SUBAPPLICATION Uebung_10c4 (* SoftKey_F1/_F2 auf DigitalOutput_Q1/_Q2 mit GreenWhiteBackground mit Typed Subapp *)
  (* Standard: 61499-2; Description: Copyright (c) 2023 Meisterschulen am Ostbahnhof This program and the accompanying materials are made available under the terms of the Eclipse Public License 2.0 which is available at https://www.eclipse.org/legal/epl-2.0/ SPDX-License-Identifier: EPL-2.0 *)
  (* Version 1.0, 2023-10-23, Franz Höpfinger, Meisterschulen am Ostbahnhof *)
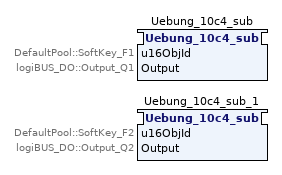
  SUBAPPS
    Uebung_10c4_sub : Uebung_10c4_sub(u16ObjId := DefaultPool::SoftKey_F1, Output := logiBUS_DO::Output_Q1);
    Uebung_10c4_sub_1 : Uebung_10c4_sub(u16ObjId := DefaultPool::SoftKey_F2, Output := logiBUS_DO::Output_Q2);
  END_SUBAPPS
END_SUBAPPLICATION
